PROGRAM MAIN
VAR
	(**)
	fbGame			: FB_Game;
	(*Button*)
	btStart			: BOOL;
	btPause			: BOOL;
	(*State*)
	GameRunning			: BOOL;
END_VAR

IF btStart THEN
	btStart := NOT btStart;
	GameRunning := TRUE;
END_IF

IF btPause THEN
	btPause := NOT btPause;
	GameRunning := FALSE;
END_IF

IF GameRunning THEN
	fbGame();
END_IF

END_PROGRAM

(* stored: Version 1.1.0.1, ProductVersion 3.1.4024.12
   POU MAIN: Id {04ca34de-edc0-468b-a7f7-08b20ad2d003}, SpecialFunc None *)
